TYPE ST_GCodeInfo2 :
STRUCT
		nTargetObjId			: UINT;		//Für mehrere Slides auf dem Target: beim GCode Start soll richtiges Target ausgewählt werden -> Target über OBJId identifiziert
END_STRUCT
END_TYPE

(* stored: Version 1.1.0.1, ProductVersion 3.1.4024.15
   DUT ST_GCodeInfo2: Id {1efabd5d-a247-4244-a5b2-5bcc9fd05d41} *)
